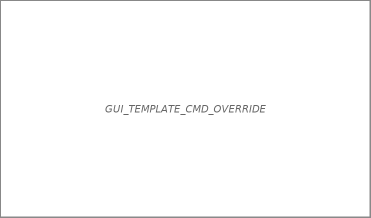
VISUALIZATION GUI_CMD_OVERRIDE  // 371x218
    Frame (0,0 371x218)
        shows GUI_TEMPLATE_CMD_OVERRIDE(m_Cmd := MAIN.cmdOverrideTest)
END_VISUALIZATION

(* stored: Version 1.1.0.1, ProductVersion 3.1.4024.12
   Visu GUI_CMD_OVERRIDE: Id {aade0da1-b953-4af5-8afd-0421f05b9631} *)
